// TwinCAT 3 PLC project LoggingExample
// ProgramVersion: 3.1.4023.0
// libraries:
//   Tc2_Standard, * (Beckhoff Automation GmbH)
//   Tc2_System, * (Beckhoff Automation GmbH)
//   Tc2_Utilities, * (Beckhoff Automation GmbH)
//   Tc3_Module, * (Beckhoff Automation GmbH)
//   Log4TC,0.0.1,mbc engineering GmbH
// project tree:
//   / F_ReadSimulatedTemperature.TcPOU, MAIN.TcPOU, PlcTask.TcTTO
// real-time tasks:
//   TASK PlcTask: cycle T#10ms, priority 20, ADS port 350

CONFIGURATION LoggingExample
    RESOURCE PLC ON TwinCAT3
        TASK PlcTask(INTERVAL := T#10ms, PRIORITY := 20);
        PROGRAM MAIN WITH PlcTask : MAIN;
    END_RESOURCE
END_CONFIGURATION

// ---- MAIN.TcPOU
PROGRAM MAIN
VAR
	fbIntervalTimer		: tc2_standard.TON := (PT:=T#5S);
	fTempRoom			: LREAL;
	nOnlineChangeCnt	: UDINT;
END_VAR

// Example 1: Cyclic logging of some values
fbIntervalTimer(IN:=NOT fbIntervalTimer.Q);
IF fbIntervalTimer.Q THEN
	fTempRoom := F_ReadSimulatedTemperature();
	
	// Log the temperature to log4tc system. Use the function
	// with logger name and one ANY argument.
	log4tc.F_LogLA1(
		E_LogLevel.eInfo,
		'MAIN',
		'Room temperature {roomTemp} °C',
		fTempRoom
	);
END_IF

// Example 2: Event based logging
IF _TaskInfo[Tc2_System.GETCURTASKINDEXEX()].FirstCycle THEN
	// Log the plc start to the log4tc system.
	log4tc.F_LogLA1(E_LogLevel.eDebug, 'MAIN', 'PLC started with application {appName}.', _AppInfo.AppName);
END_IF

IF _AppInfo.OnlineChangeCnt <> nOnlineChangeCnt THEN
	log4tc.F_LogLA1(E_LogLevel.eInfo, 'MAIN', 'Online change executed: {changeCount}.', _AppInfo.OnlineChangeCnt);
END_IF
nOnlineChangeCnt := _AppInfo.OnlineChangeCnt;

IF _AppInfo.BSODOccured THEN
	log4tc.F_LogL(E_LogLevel.eFatal, 'MAIN', 'Windows crashed');
END_IF

// Must be called in each task, preferable once a cycle
PRG_TaskLog.Call();

END_PROGRAM

// ---- F_ReadSimulatedTemperature.TcPOU
FUNCTION F_ReadSimulatedTemperature : LREAL
VAR_STAT
	fbRand		: DRAND := (Seed:=TIME_TO_INT(TIME()));
END_VAR

fbRand();
F_ReadSimulatedTemperature := 20 + (fbRand.Num - 0.5) * 5;

END_FUNCTION
